(* IEC 61131-3 sources: ICS-simulation/services/openplc/configs, 5 files *)

(* ---- plc.st ---- *)
TYPE
  LOGLEVEL : (CRITICAL, WARNING, INFO, DEBUG) := INFO;
END_TYPE

FUNCTION_BLOCK LOGGER
  VAR_INPUT
    TRIG : BOOL;
    MSG : STRING;
    LEVEL : LOGLEVEL := INFO;
  END_VAR
  VAR
    TRIG0 : BOOL;
  END_VAR

  IF TRIG AND NOT TRIG0 THEN
  {{
   LogMessage(GetFbVar(LEVEL),(char*)GetFbVar(MSG, .body),GetFbVar(MSG, .len));
  }}
  END_IF;
  TRIG0:=TRIG;
END_FUNCTION_BLOCK

FUNCTION_BLOCK python_eval
  VAR_INPUT
    TRIG : BOOL;
    CODE : STRING;
  END_VAR
  VAR_OUTPUT
    ACK : BOOL;
    RESULT : STRING;
  END_VAR
  VAR
    STATE : DWORD;
    BUFFER : STRING;
    PREBUFFER : STRING;
    TRIGM1 : BOOL;
    TRIGGED : BOOL;
  END_VAR

  {extern void __PythonEvalFB(int, PYTHON_EVAL*);__PythonEvalFB(0, data__);}
END_FUNCTION_BLOCK

FUNCTION_BLOCK python_poll
  VAR_INPUT
    TRIG : BOOL;
    CODE : STRING;
  END_VAR
  VAR_OUTPUT
    ACK : BOOL;
    RESULT : STRING;
  END_VAR
  VAR
    STATE : DWORD;
    BUFFER : STRING;
    PREBUFFER : STRING;
    TRIGM1 : BOOL;
    TRIGGED : BOOL;
  END_VAR

  {extern void __PythonEvalFB(int, PYTHON_EVAL*);__PythonEvalFB(1,(PYTHON_EVAL*)(void*)data__);}
END_FUNCTION_BLOCK

FUNCTION_BLOCK python_gear
  VAR_INPUT
    N : UINT;
    TRIG : BOOL;
    CODE : STRING;
  END_VAR
  VAR_OUTPUT
    ACK : BOOL;
    RESULT : STRING;
  END_VAR
  VAR
    py_eval : python_eval;
    COUNTER : UINT;
    ADD10_OUT : UINT;
    EQ13_OUT : BOOL;
    SEL15_OUT : UINT;
    AND7_OUT : BOOL;
  END_VAR

  ADD10_OUT := ADD(COUNTER, 1);
  EQ13_OUT := EQ(N, ADD10_OUT);
  SEL15_OUT := SEL(EQ13_OUT, ADD10_OUT, 0);
  COUNTER := SEL15_OUT;
  AND7_OUT := AND(EQ13_OUT, TRIG);
  py_eval(TRIG := AND7_OUT, CODE := CODE);
  ACK := py_eval.ACK;
  RESULT := py_eval.RESULT;
END_FUNCTION_BLOCK

PROGRAM program0
  VAR
    inputA : BOOL;
    inputB : BOOL;
    outputAND : BOOL;
    outputOR : BOOL;
  END_VAR

  outputAND := inputB AND inputA;
  outputOR := inputA OR inputB;
END_PROGRAM

CONFIGURATION Config0

  RESOURCE Res0 ON PLC
    TASK task0(INTERVAL := T#20ms,PRIORITY := 0);
    PROGRAM instance0 WITH task0 : program0;
  END_RESOURCE
END_CONFIGURATION

(* ---- led.st ---- *)
PROGRAM led_switch
  VAR
    PB1 AT %IX200.0 : BOOL;
    PB2 AT %IX200.1 : BOOL;
    LED AT %QX200.0 : BOOL;
  END_VAR

  LED := NOT(PB2) AND (LED OR PB1);
END_PROGRAM

CONFIGURATION Config0

  RESOURCE Res0 ON PLC
    TASK task0(INTERVAL := T#20ms,PRIORITY := 0);
    PROGRAM instance0 WITH task0 : led_switch;
  END_RESOURCE
END_CONFIGURATION

(* ---- led2.st ---- *)
PROGRAM led_switch
  VAR
    PB1 AT %IX100.0 : BOOL;
    PB2 AT %IX100.1 : BOOL;
    LED AT %QX100.0 : BOOL;
  END_VAR

  LED := NOT(PB2) AND (LED OR PB1);
END_PROGRAM

CONFIGURATION Config0

  RESOURCE Res0 ON PLC
    TASK task0(INTERVAL := T#20ms,PRIORITY := 0);
    PROGRAM instance0 WITH task0 : led_switch;
  END_RESOURCE
END_CONFIGURATION

(* ---- mixer.st ---- *)
PROGRAM OB1
  VAR
    TANK_LLS AT %QX100.4 : BOOL;
    TANK_HLS AT %QX100.5 : BOOL;
    STOP AT %QX100.6 : BOOL;
  END_VAR
  VAR
    ELAPSED_TIME : TIME;
  END_VAR
  VAR
    PUMP_A AT %QX100.0 : BOOL;
    PUMP_B AT %QX100.1 : BOOL;
    MIXER AT %QX100.2 : BOOL;
    VALVE AT %QX100.3 : BOOL;
  END_VAR
  VAR
    SR0 : SR;
    TP0 : TP;
    SR1 : SR;
  END_VAR
  VAR
    IntTime AT %MW0 : INT := 5;
  END_VAR
  VAR
    INT_TO_TIME44_OUT : TIME;
  END_VAR

  SR0(S1 := TANK_LLS, R := NOT(STOP) OR TANK_HLS);
  PUMP_A := SR0.Q1;
  PUMP_B := SR0.Q1;
  INT_TO_TIME44_OUT := INT_TO_TIME(IntTime);
  TP0(IN := NOT(VALVE) AND TANK_HLS, PT := INT_TO_TIME44_OUT);
  MIXER := TP0.Q;
  ELAPSED_TIME := TP0.ET;
  SR1(S1 := NOT(MIXER) AND TANK_HLS, R := NOT(STOP) OR TANK_LLS);
  VALVE := SR1.Q1;
END_PROGRAM

CONFIGURATION Config0

  RESOURCE Res0 ON PLC
    TASK task0(INTERVAL := T#20ms,PRIORITY := 0);
    PROGRAM instance0 WITH task0 : OB1;
  END_RESOURCE
END_CONFIGURATION

(* ---- water_tank.st ---- *)
PROGRAM program0
  VAR
    Pool_LLS AT %IX100 : BOOL;
    Tank_LLS AT %IX101 : BOOL;
    Tank_HLS AT %IX102 : BOOL;
    Motor_ON AT %QX100 : BOOL;
  END_VAR
  VAR
    SR0 : SR;
  END_VAR

  SR0(S1 := NOT(Tank_LLS), R := NOT(Pool_LLS) OR Tank_HLS);
  Motor_ON := SR0.Q1;
END_PROGRAM

CONFIGURATION Config0

  RESOURCE Res0 ON PLC
    TASK task0(INTERVAL := T#20ms,PRIORITY := 0);
    PROGRAM instance0 WITH task0 : program0;
  END_RESOURCE
END_CONFIGURATION
